PROGRAM IO_SWITCHBOARD
VAR CONSTANT
	STATE_TIMEOUT : INT := 10;
END_VAR
VAR
	state : SYSTEM_STATE;
	stateIdleCounter : INT;
	isConsoleActive : BOOL;
	isRemoteActive : BOOL;
	
	CONSOLE_DOWN_BUTTON_IN AT %I* : BOOL;
	CONSOLE_RUN_BUTTON_IN AT %I* : BOOL;
	CONSOLE_UP_BUTTON_IN AT %I* : BOOL;
	
	REMOTE_DOWN_BUTTON_IN AT %I* : BOOL;
	REMOTE_RUN_BUTTON_IN AT %I* : BOOL;
	REMOTE_UP_BUTTON_IN AT %I* : BOOL;
END_VAR

isConsoleActive := (CONSOLE_DOWN_BUTTON_IN OR CONSOLE_RUN_BUTTON_IN OR CONSOLE_UP_BUTTON_IN);
isRemoteActive := (REMOTE_DOWN_BUTTON_IN OR REMOTE_RUN_BUTTON_IN OR REMOTE_UP_BUTTON_IN);

CASE state OF 
	SYSTEM_STATE.SYSTEM_READY :
		GV_LIFT.CONSOLE_ACTIVE_INDICATOR_OUT := FALSE;
		GV_LIFT.REMOTE_ACTIVE_INDICATOR_OUT := FALSE;
		IF isConsoleActive THEN
			state := SYSTEM_STATE.CONSOLE_CONTROL;
		ELSIF isRemoteActive THEN
			state := SYSTEM_STATE.REMOTE_CONTROL;
		END_IF
		
	SYSTEM_STATE.CONSOLE_CONTROL :
		IF isConsoleActive THEN
			IF CONSOLE_RUN_BUTTON_IN THEN
				GV_LIFT.RUN_BUTTON_OUT := CONSOLE_RUN_BUTTON_IN;
			ELSE
				GV_LIFT.DOWN_BUTTON_OUT := CONSOLE_DOWN_BUTTON_IN;
				GV_LIFT.UP_BUTTON_OUT := CONSOLE_UP_BUTTON_IN;
			END_IF
			stateIdleCounter := 0;
			GV_LIFT.CONSOLE_ACTIVE_INDICATOR_OUT := TRUE;
		ELSE
			stateIdleCounter := stateIdleCounter + 1;
			IF(stateIdleCounter >= STATE_TIMEOUT) THEN
				stateIdleCounter := 0;
				state := SYSTEM_STATE.SYSTEM_READY;
			END_IF
		END_IF
		
		SYSTEM_STATE.REMOTE_CONTROL :
		IF isRemoteActive THEN
			IF REMOTE_RUN_BUTTON_IN THEN
				GV_LIFT.RUN_BUTTON_OUT := REMOTE_RUN_BUTTON_IN;
			ELSE
				GV_LIFT.DOWN_BUTTON_OUT := REMOTE_DOWN_BUTTON_IN;
				GV_LIFT.UP_BUTTON_OUT := REMOTE_UP_BUTTON_IN;
			END_IF
			stateIdleCounter := 0;
			GV_LIFT.REMOTE_ACTIVE_INDICATOR_OUT := TRUE;
		ELSE
			stateIdleCounter := stateIdleCounter + 1;
			IF(stateIdleCounter >= STATE_TIMEOUT) THEN
				stateIdleCounter := 0;
				state := SYSTEM_STATE.SYSTEM_READY;
			END_IF
		END_IF
END_CASE

GV_LIFT.DOWN_INDICATOR_OUT := GV_LIFT.DOWN_INDICATOR_IN;
GV_LIFT.UP_INDICATOR_OUT := GV_LIFT.UP_INDICATOR_IN;

GV_LIFT.CRUSH_PROTECTION_INDICATOR_OUT := NOT GV_LIFT.CRUSH_PROTECTION_INDICATOR_IN;

GV_LIFT.DOWNSTAGE_ESTOP_INDICATOR_OUT := NOT GV_LIFT.DOWNSTAGE_ESTOP_INDICATOR_IN;
GV_LIFT.UPSTAGE_ESTOP_INDICATOR_OUT := NOT GV_LIFT.UPSTAGE_ESTOP_INDICATOR_IN;
GV_LIFT.REMOTE_ESTOP_INDICATOR_OUT := NOT GV_LIFT.REMOTE_ESTOP_INDICATOR_IN;
GV_LIFT.PIT_ESTOP_INDICATOR_OUT := NOT GV_LIFT.PIT_ESTOP_INDICATOR_IN;
GV_LIFT.CONSOLE_ESTOP_INDICATOR_OUT := NOT GV_LIFT.CONSOLE_ESTOP_INDICATOR_IN;
GV_LIFT.PUMP_ESTOP_INDICATOR_OUT := NOT GV_LIFT.PUMP_ESTOP_INDICATOR_IN;

GV_LIFT.ESTOP_INDICATOR_OUT := GV_LIFT.ESTOP_INDICATOR_IN;

GV_LIFT.DOOR_1_INDICATOR_OUT := NOT GV_LIFT.DOOR_1_INDICATOR_IN;
GV_LIFT.DOOR_1_INDICATOR_LATCH_OUT := NOT GV_LIFT.DOOR_1_INDICATOR_LATCH_OUT;
GV_LIFT.DOOR_2_INDICATOR_OUT := NOT GV_LIFT.DOOR_2_INDICATOR_IN;
GV_LIFT.DOOR_2_INDICATOR_LATCH_OUT := NOT GV_LIFT.DOOR_2_INDICATOR_LATCH_OUT;
GV_LIFT.DOOR_3_INDICATOR_OUT := NOT GV_LIFT.DOOR_3_INDICATOR_IN;
GV_LIFT.DOOR_3_INDICATOR_LATCH_OUT := NOT GV_LIFT.DOOR_3_INDICATOR_LATCH_OUT;
GV_LIFT.DOOR_4_INDICATOR_OUT := NOT GV_LIFT.DOOR_4_INDICATOR_IN;
GV_LIFT.DOOR_4_INDICATOR_LATCH_OUT := NOT GV_LIFT.DOOR_4_INDICATOR_LATCH_OUT;

GV_LIFT.UP_LIMIT_INDICATOR_OUT := NOT GV_LIFT.UP_LIMIT_INDICATOR_IN;
GV_LIFT.UP_LIMIT_INDICATOR_LATCH_OUT := NOT GV_LIFT.UP_LIMIT_INDICATOR_LATCH_IN;
GV_LIFT.DOWN_LIMIT_INDICATOR_OUT := NOT GV_LIFT.DOWN_LIMIT_INDICATOR_IN;
GV_LIFT.DOWN_LIMIT_INDICATOR_LATCH_OUT := NOT GV_LIFT.DOWN_LIMIT_INDICATOR_LATCH_IN;
GV_LIFT.ULTIMATE_LIMIT_INDICATOR_OUT := NOT GV_LIFT.ULTIMATE_LIMIT_INDICATOR_IN;
GV_LIFT.ULTIMATE_LIMIT_INDICATOR_LATCH_OUT := NOT GV_LIFT.ULTIMATE_LIMIT_INDICATOR_LATCH_IN;

END_PROGRAM

(* stored: Version 1.1.0.1, ProductVersion 3.1.4022.12
   POU IO_SWITCHBOARD: Id {a90d9e50-84d3-4175-8411-1c95f1ec50a2}, SpecialFunc None *)
